% RSLogix 500 project P4_New.RSS, saved by version 12.00.00.00 %
PROJECT "UNTITLED"    % processor: Bul.1763 MicroLogix 1100 Series B %

PROGRAM FILES
  LAD 2   4 rungs
  LAD 3 "IO"  7 rungs
  LAD 4 "CTRL"  11 rungs
  LAD 5 "POS"  10 rungs

DATA FILES
  O0 OUTPUT  4 elements
  I1 INPUT  6 elements
  S2 STATUS  66 elements
  B3 BINARY  2 elements
  T4 TIMER  3 elements
  C5 COUNTER  1 elements
  R6 CONTROL  1 elements
  N7 INTEGER  2 elements
  F8 FLOAT  1 elements

LADDER 2
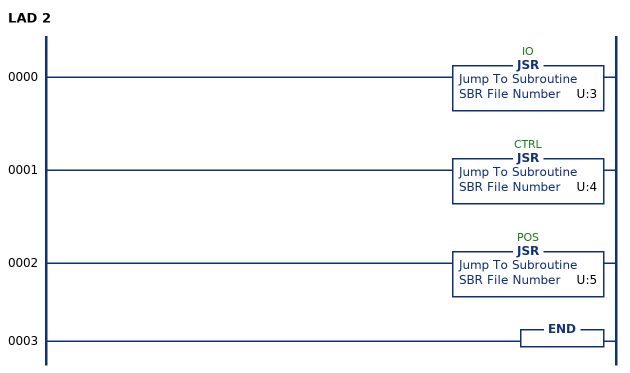
% Rung: 0 %
SOR JSR U:3 EOR
%   U:3  "IO" %
% Rung: 1 %
SOR JSR U:4 EOR
%   U:4  "CTRL" %
% Rung: 2 %
SOR JSR U:5 EOR
%   U:5  "POS" %
% Rung: 3 %
SOR END EOR

LADDER 3 "IO"
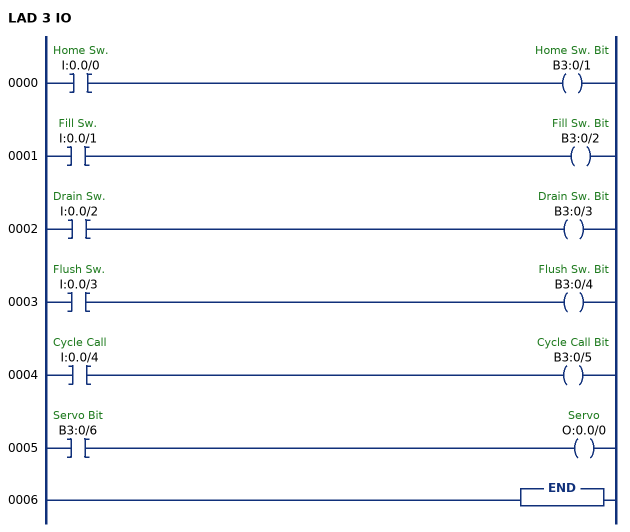
% Rung: 0 %
SOR XIC I:0.0/0 OTE B3:0/1 EOR
%   I:0.0/0  "Home Sw." %
%   B3:0/1  "Home Sw. Bit" %
% Rung: 1 %
SOR XIC I:0.0/1 OTE B3:0/2 EOR
%   I:0.0/1  "Fill Sw." %
%   B3:0/2  "Fill Sw. Bit" %
% Rung: 2 %
SOR XIC I:0.0/2 OTE B3:0/3 EOR
%   I:0.0/2  "Drain Sw." %
%   B3:0/3  "Drain Sw. Bit" %
% Rung: 3 %
SOR XIC I:0.0/3 OTE B3:0/4 EOR
%   I:0.0/3  "Flush Sw." %
%   B3:0/4  "Flush Sw. Bit" %
% Rung: 4 %
SOR XIC I:0.0/4 OTE B3:0/5 EOR
%   I:0.0/4  "Cycle Call" %
%   B3:0/5  "Cycle Call Bit" %
% Rung: 5 %
SOR XIC B3:0/6 OTE O:0.0/0 EOR
%   B3:0/6  "Servo Bit" %
%   O:0.0/0  "Servo" %
% Rung: 6 %
SOR END EOR

LADDER 4 "CTRL"
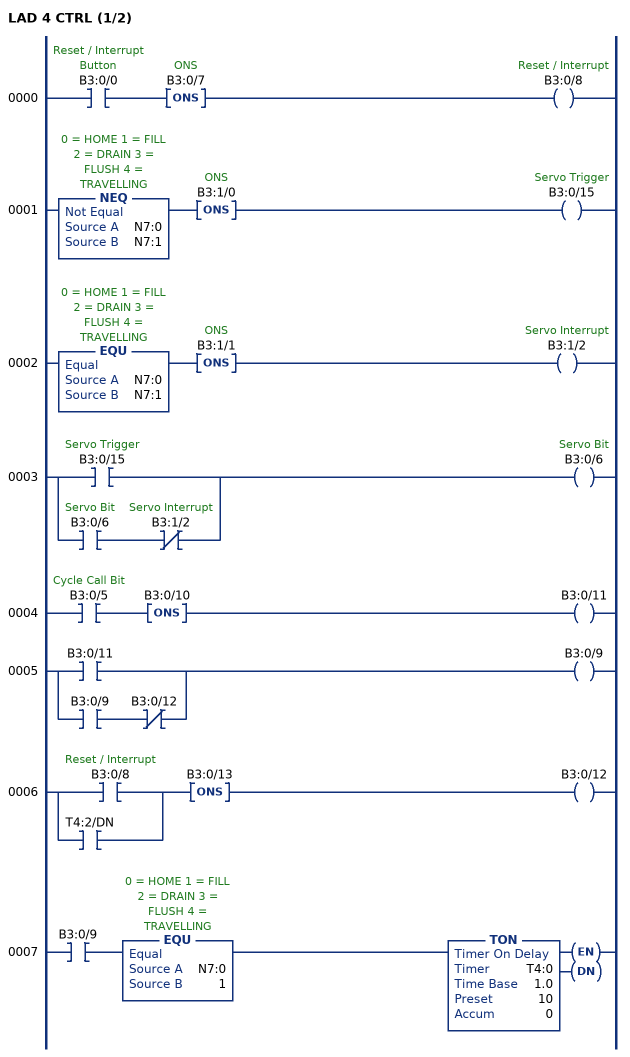
% Rung: 0 %
SOR XIC B3:0/0 ONS B3:0/7 OTE B3:0/8 EOR
%   B3:0/0  "Reset / Interrupt Button" %
%   B3:0/7  "ONS" %
%   B3:0/8  "Reset / Interrupt" %
% Rung: 1 %
SOR NEQ N7:0 N7:1 ONS B3:1/0 OTE B3:0/15 EOR
%   N7:0  "0 = HOME 1 = FILL 2 = DRAIN 3 = FLUSH 4 = TRAVELLING" %
%   N7:1  "Desired: 0 = HOME 1 = FILL 2 = DRAIN 3 = FLUSH" %
%   B3:1/0  "ONS" %
%   B3:0/15  "Servo Trigger" %
% Rung: 2 %
SOR EQU N7:0 N7:1 ONS B3:1/1 OTE B3:1/2 EOR
%   N7:0  "0 = HOME 1 = FILL 2 = DRAIN 3 = FLUSH 4 = TRAVELLING" %
%   N7:1  "Desired: 0 = HOME 1 = FILL 2 = DRAIN 3 = FLUSH" %
%   B3:1/1  "ONS" %
%   B3:1/2  "Servo Interrupt" %
% Rung: 3 %
SOR BST XIC B3:0/15 NXB XIC B3:0/6 XIO B3:1/2 BND OTE B3:0/6 EOR
%   B3:0/15  "Servo Trigger" %
%   B3:0/6  "Servo Bit" %
%   B3:1/2  "Servo Interrupt" %
% Rung: 4 %
SOR XIC B3:0/5 ONS B3:0/10 OTE B3:0/11 EOR
%   B3:0/5  "Cycle Call Bit" %
% Rung: 5 %
SOR BST XIC B3:0/11 NXB XIC B3:0/9 XIO B3:0/12 BND OTE B3:0/9 EOR
% Rung: 6 %
SOR BST XIC B3:0/8 NXB XIC T4:2/DN BND ONS B3:0/13 OTE B3:0/12 EOR
%   B3:0/8  "Reset / Interrupt" %
% Rung: 7 %
SOR XIC B3:0/9 EQU N7:0 1 TON T4:0 1.0 10 0 EOR
%   N7:0  "0 = HOME 1 = FILL 2 = DRAIN 3 = FLUSH 4 = TRAVELLING" %

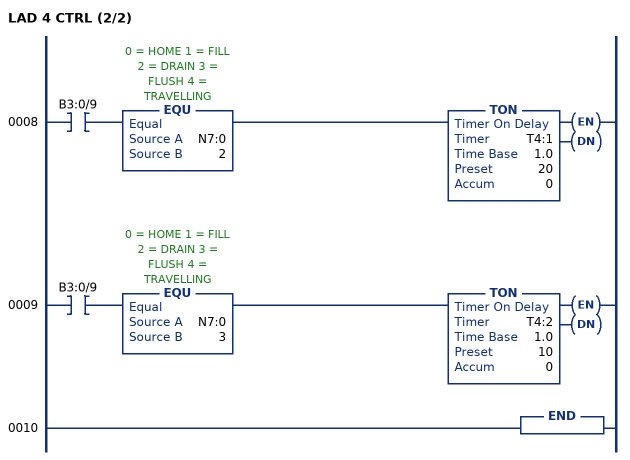
% Rung: 8 %
SOR XIC B3:0/9 EQU N7:0 2 TON T4:1 1.0 20 0 EOR
%   N7:0  "0 = HOME 1 = FILL 2 = DRAIN 3 = FLUSH 4 = TRAVELLING" %
% Rung: 9 %
SOR XIC B3:0/9 EQU N7:0 3 TON T4:2 1.0 10 0 EOR
%   N7:0  "0 = HOME 1 = FILL 2 = DRAIN 3 = FLUSH 4 = TRAVELLING" %
% Rung: 10 %
SOR END EOR

LADDER 5 "POS"
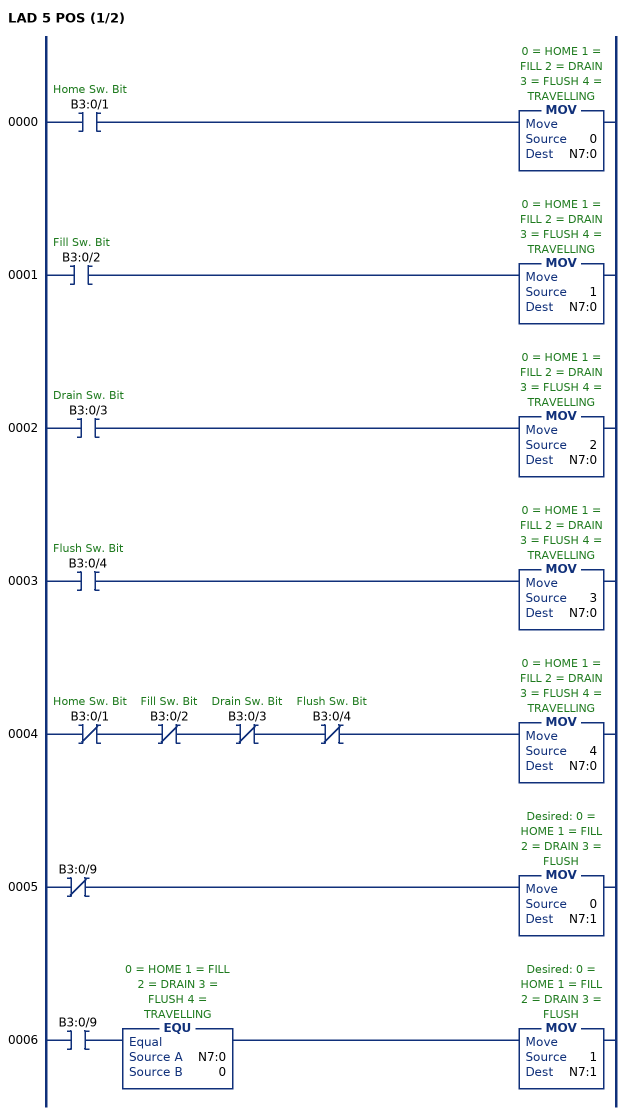
% Rung: 0 %
SOR XIC B3:0/1 MOV 0 N7:0 EOR
%   B3:0/1  "Home Sw. Bit" %
%   N7:0  "0 = HOME 1 = FILL 2 = DRAIN 3 = FLUSH 4 = TRAVELLING" %
% Rung: 1 %
SOR XIC B3:0/2 MOV 1 N7:0 EOR
%   B3:0/2  "Fill Sw. Bit" %
%   N7:0  "0 = HOME 1 = FILL 2 = DRAIN 3 = FLUSH 4 = TRAVELLING" %
% Rung: 2 %
SOR XIC B3:0/3 MOV 2 N7:0 EOR
%   B3:0/3  "Drain Sw. Bit" %
%   N7:0  "0 = HOME 1 = FILL 2 = DRAIN 3 = FLUSH 4 = TRAVELLING" %
% Rung: 3 %
SOR XIC B3:0/4 MOV 3 N7:0 EOR
%   B3:0/4  "Flush Sw. Bit" %
%   N7:0  "0 = HOME 1 = FILL 2 = DRAIN 3 = FLUSH 4 = TRAVELLING" %
% Rung: 4 %
SOR XIO B3:0/1 XIO B3:0/2 XIO B3:0/3 XIO B3:0/4 MOV 4 N7:0 EOR
%   B3:0/1  "Home Sw. Bit" %
%   B3:0/2  "Fill Sw. Bit" %
%   B3:0/3  "Drain Sw. Bit" %
%   B3:0/4  "Flush Sw. Bit" %
%   N7:0  "0 = HOME 1 = FILL 2 = DRAIN 3 = FLUSH 4 = TRAVELLING" %
% Rung: 5 %
SOR XIO B3:0/9 MOV 0 N7:1 EOR
%   N7:1  "Desired: 0 = HOME 1 = FILL 2 = DRAIN 3 = FLUSH" %
% Rung: 6 %
SOR XIC B3:0/9 EQU N7:0 0 MOV 1 N7:1 EOR
%   N7:0  "0 = HOME 1 = FILL 2 = DRAIN 3 = FLUSH 4 = TRAVELLING" %
%   N7:1  "Desired: 0 = HOME 1 = FILL 2 = DRAIN 3 = FLUSH" %

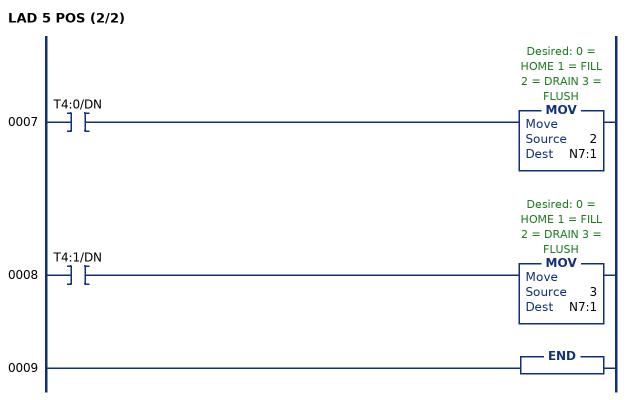
% Rung: 7 %
SOR XIC T4:0/DN MOV 2 N7:1 EOR
%   N7:1  "Desired: 0 = HOME 1 = FILL 2 = DRAIN 3 = FLUSH" %
% Rung: 8 %
SOR XIC T4:1/DN MOV 3 N7:1 EOR
%   N7:1  "Desired: 0 = HOME 1 = FILL 2 = DRAIN 3 = FLUSH" %
% Rung: 9 %
SOR END EOR

DATA TABLE (non-zero values as saved)
DATA T4
% .PRE .ACC %
% T4:0 % 10 0
% T4:1 % 20 0
% T4:2 % 10 0
